Fanuc KAREL source: kt00726.KL

-- PROVISIONAL review KL for V940-1; original PC SHA256 1f701ae59b414f1d221cdae51184ab46e10671347cf65f497efde405923b76cb
-- Incomplete behavior may be omitted. Consult companion uncertainty JSON. Do not deploy.
PROGRAM KT00726
%NOLOCKGROUP
VAR
  OUT : BOOLEAN
-- UNRESOLVED_DECL V1 type=000013
-- UNRESOLVED_DECL V2 type=000013
BEGIN
  -- V9_ZERO_TABLE_METADATA_HINT layout=0001; no indexed target words; source/name/runtime held
  -- UNRESOLVED_PC offsets 5-20; opcodes 2E,22,32,35
  -- UNRESOLVED_PC offsets 25-40; opcodes 2E,22,32,35
  -- UNRESOLVED_PC offsets 45-60; opcodes 2E,22,32,35
  -- UNRESOLVED_PC offsets 65-80; opcodes 2E,22,32,35
  -- UNRESOLVED_PC offsets 85-100; opcodes 22,63,23
  -- UNRESOLVED_PC offsets 105-109; opcodes 7F
END KT00726
